PROGRAM PRG_2_PMPS
VAR
END_VAR

END_PROGRAM

(* stored: Version 1.1.0.1, ProductVersion 3.1.4022.12
   POU PRG_2_PMPS: Id {2f4e980b-04a5-4967-a693-b70eb29ff6ac}, SpecialFunc None *)
